TYPE ST_System_MVHW_Steuerung :
STRUCT
	Freigabe				: ST_Steuerung_auto_manu_BOOL;
	Freigabe_Deakt		: ST_Steuerung_auto_manu_BOOL;
	Betrieb_Anford		: ST_Steuerung_auto_manu_opti_BOOL;



	Quittierung			: BOOL;
END_STRUCT
END_TYPE

(* stored: Version 1.1.0.1, ProductVersion 3.1.4024.9
   DUT ST_System_MVHW_Steuerung: Id {d48a75f3-98bc-403a-8aa9-849e5cc4e698} *)
